FUNCTION A_UINT : ST_Arg
VAR_INPUT
	nNumber	: REFERENCE TO UINT;
END_VAR

IF __ISVALIDREF(nNumber) THEN
	A_UINT.eType := E_ArgType.UIntArg;
	A_UINT.pData := ADR(nNumber);
	A_UINT.nSize := SIZEOF(UINT);
END_IF

END_FUNCTION

(* stored: Version 1.1.0.1, ProductVersion 3.1.4024.15
   POU A_UINT: Id {8dffa0f8-924c-435b-b298-f3b79daefb8e}, SpecialFunc None *)
